(* PLC project PLC, Beckhoff Automation GmbH TwinCAT PLC Control 3.5.20.60 *)
(* stored: creationDateTime 2026-07-21T08:44:28.1635996, modificationDateTime 2026-07-21T08:44:28.1635996 *)

TYPE ST_ADS_API_ScadaViewerApp_PLC_Out :

STRUCT

	Status				:	ST_ADS_API_ScadaViewerApp_PLC_Out_Status;	// |1| Status PLC aplikace
	
END_STRUCT

END_TYPE
